// TIA Portal V19 export
DATA_BLOCK "InstLiftSeq"   // DB12
TITLE = InstLiftSeq
{ DB_Accessible_From_OPC_UA := 'FALSE' }
// IDB LiftSeq
// stored: DBAccessibleFromOPCUA false, InstanceOfName LiftSeq, InstanceOfType FB
"LiftSeq"
   // // inherited from GRAPH_BASE
   // VAR_INPUT
   //    OFF_SQ { ExternalWritable := 'False'} : Bool;
   //    INIT_SQ { ExternalWritable := 'False'} : Bool;
   //    ACK_EF { ExternalWritable := 'False'} : Bool;
   //    REG_EF { ExternalWritable := 'False'} : Bool;
   //    ACK_S { ExternalWritable := 'False'} : Bool;
   //    REG_S { ExternalWritable := 'False'} : Bool;
   //    HALT_SQ { ExternalWritable := 'False'} : Bool;
   //    HALT_TM { ExternalWritable := 'False'} : Bool;
   //    ZERO_OP { ExternalWritable := 'False'} : Bool;
   //    EN_IL { ExternalWritable := 'False'} : Bool;
   //    EN_SV { ExternalWritable := 'False'} : Bool;
   //    EN_ACKREQ { ExternalWritable := 'False'} : Bool;
   //    EN_SSKIP { ExternalWritable := 'False'} : Bool;
   //    DISP_SACT { ExternalWritable := 'False'} : Bool;
   //    DISP_SEF { ExternalWritable := 'False'} : Bool;
   //    DISP_SALL { ExternalWritable := 'False'} : Bool;
   //    S_PREV { ExternalWritable := 'False'} : Bool;
   //    S_NEXT { ExternalWritable := 'False'} : Bool;
   //    SW_AUTO { ExternalWritable := 'False'} : Bool;
   //    SW_TAP { ExternalWritable := 'False'} : Bool;
   //    SW_TOP { ExternalWritable := 'False'} : Bool;
   //    SW_MAN { ExternalWritable := 'False'} : Bool;
   //    S_SEL { ExternalWritable := 'False'} : Int;
   //    S_SELOK { ExternalWritable := 'False'} : Bool;
   //    S_ON { ExternalWritable := 'False'} : Bool;
   //    S_OFF { ExternalWritable := 'False'} : Bool;
   //    T_PREV { ExternalWritable := 'False'} : Bool;
   //    T_NEXT { ExternalWritable := 'False'} : Bool;
   //    T_PUSH { ExternalWritable := 'False'} : Bool;
   //    EN_LMODE { ExternalWritable := 'False'} : Bool;
   //    RESET_CRIT { ExternalWritable := 'False'} : Bool;
   // END_VAR
   // VAR_OUTPUT
   //    S_NO { ExternalWritable := 'False'} : Int;
   //    S_MORE { ExternalWritable := 'False'} : Bool;
   //    S_ACTIVE { ExternalWritable := 'False'} : Bool;
   //    S_TIME { ExternalWritable := 'False'} : Time;
   //    S_TIMEOK { ExternalWritable := 'False'} : Time;
   //    S_CRITLOC { ExternalWritable := 'False'} : DWord;
   //    S_CRITLOCERR { ExternalWritable := 'False'} : DWord;
   //    S_STATE { ExternalWritable := 'False'} : Word;
   //    T_NO { ExternalWritable := 'False'} : Int;
   //    T_MORE { ExternalWritable := 'False'} : Bool;
   //    T_CRIT { ExternalWritable := 'False'} : DWord;
   //    T_CRITOLD { ExternalWritable := 'False'} : DWord;
   //    T_CRITFLT { ExternalWritable := 'False'} : DWord;
   //    ERROR { ExternalWritable := 'False'} : Bool;
   //    FAULT { ExternalWritable := 'False'} : Bool;
   //    ERR_FLT { ExternalWritable := 'False'} : Bool;
   //    SQ_ISOFF { ExternalWritable := 'False'} : Bool;
   //    SQ_HALTED { ExternalWritable := 'False'} : Bool;
   //    TM_HALTED { ExternalWritable := 'False'} : Bool;
   //    OP_ZEROED { ExternalWritable := 'False'} : Bool;
   //    IL_ENABLED { ExternalWritable := 'False'} : Bool;
   //    SV_ENABLED { ExternalWritable := 'False'} : Bool;
   //    ACKREQ_ENABLED { ExternalWritable := 'False'} : Bool;
   //    SSKIP_ENABLED { ExternalWritable := 'False'} : Bool;
   //    SACT_DISP { ExternalWritable := 'False'} : Bool;
   //    SEF_DISP { ExternalWritable := 'False'} : Bool;
   //    SALL_DISP { ExternalWritable := 'False'} : Bool;
   //    AUTO_ON { ExternalWritable := 'False'} : Bool;
   //    TAP_ON { ExternalWritable := 'False'} : Bool;
   //    TOP_ON { ExternalWritable := 'False'} : Bool;
   //    MAN_ON { ExternalWritable := 'False'} : Bool;
   //    LMODE_ENABLED { ExternalWritable := 'False'} : Bool;
   // END_VAR
   // VAR RETAIN
   //    RT_DATA { ExternalWritable := 'False'; S7_SetPoint := 'True'} : G7_RTDataPlus_V6;
   //    "Start band" { ExternalWritable := 'False'; S7_SetPoint := 'True'} : G7_TransitionPlus_V6;
   //    "Step 4 Conditions" { ExternalWritable := 'False'; S7_SetPoint := 'True'} : G7_TransitionPlus_V6;
   //    "Start of lift 1" { ExternalWritable := 'False'; S7_SetPoint := 'True'} : G7_TransitionPlus_V6;
   //    "Lift 1 up" { ExternalWritable := 'False'; S7_SetPoint := 'True'} : G7_TransitionPlus_V6;
   //    "Lift 1 down" { ExternalWritable := 'False'; S7_SetPoint := 'True'} : G7_TransitionPlus_V6;
   //    "Step 7 Conditions" { ExternalWritable := 'False'; S7_SetPoint := 'True'} : G7_TransitionPlus_V6;
   //    "Start of lift 2" { ExternalWritable := 'False'; S7_SetPoint := 'True'} : G7_TransitionPlus_V6;
   //    "Lift 2 up" { ExternalWritable := 'False'; S7_SetPoint := 'True'} : G7_TransitionPlus_V6;
   //    "Lift 2 down" { ExternalWritable := 'False'; S7_SetPoint := 'True'} : G7_TransitionPlus_V6;
   //    Init { ExternalWritable := 'False'; S7_SetPoint := 'True'} : G7_StepPlus_V6;
   //    "Deactivate Stop 1" { ExternalWritable := 'False'; S7_SetPoint := 'True'} : G7_StepPlus_V6;
   //    "Activate    Stop 2" { ExternalWritable := 'False'; S7_SetPoint := 'True'} : G7_StepPlus_V6;
   //    "Lift 1 moves up" { ExternalWritable := 'False'; S7_SetPoint := 'True'} : G7_StepPlus_V6;
   //    "Lift 1 moves down" { ExternalWritable := 'False'; S7_SetPoint := 'True'} : G7_StepPlus_V6;
   //    "Deactivate Stop 2" { ExternalWritable := 'False'; S7_SetPoint := 'True'} : G7_StepPlus_V6;
   //    "Lift 2 moves up" { ExternalWritable := 'False'; S7_SetPoint := 'True'} : G7_StepPlus_V6;
   //    "Lift 2 moves down" { ExternalWritable := 'False'; S7_SetPoint := 'True'} : G7_StepPlus_V6;
   // END_VAR
BEGIN
END_DATA_BLOCK
